TYPE DriveStatus :
STRUCT
	ReadyToEnable : BOOL;
	Ready : BOOL;
	Warning : BOOL;
	Error : BOOL;
	MovingPositive : BOOL;
	MovingNegative : BOOL;
	DigitalInput1 : BOOL;
	DigitalInput2 : BOOL;
END_STRUCT
END_TYPE

(* stored: Version 1.1.0.1, ProductVersion 3.1.4024.11
   DUT DriveStatus: Id {c79d0e04-3606-438b-a8bf-2e6ccf7eb7eb} *)
